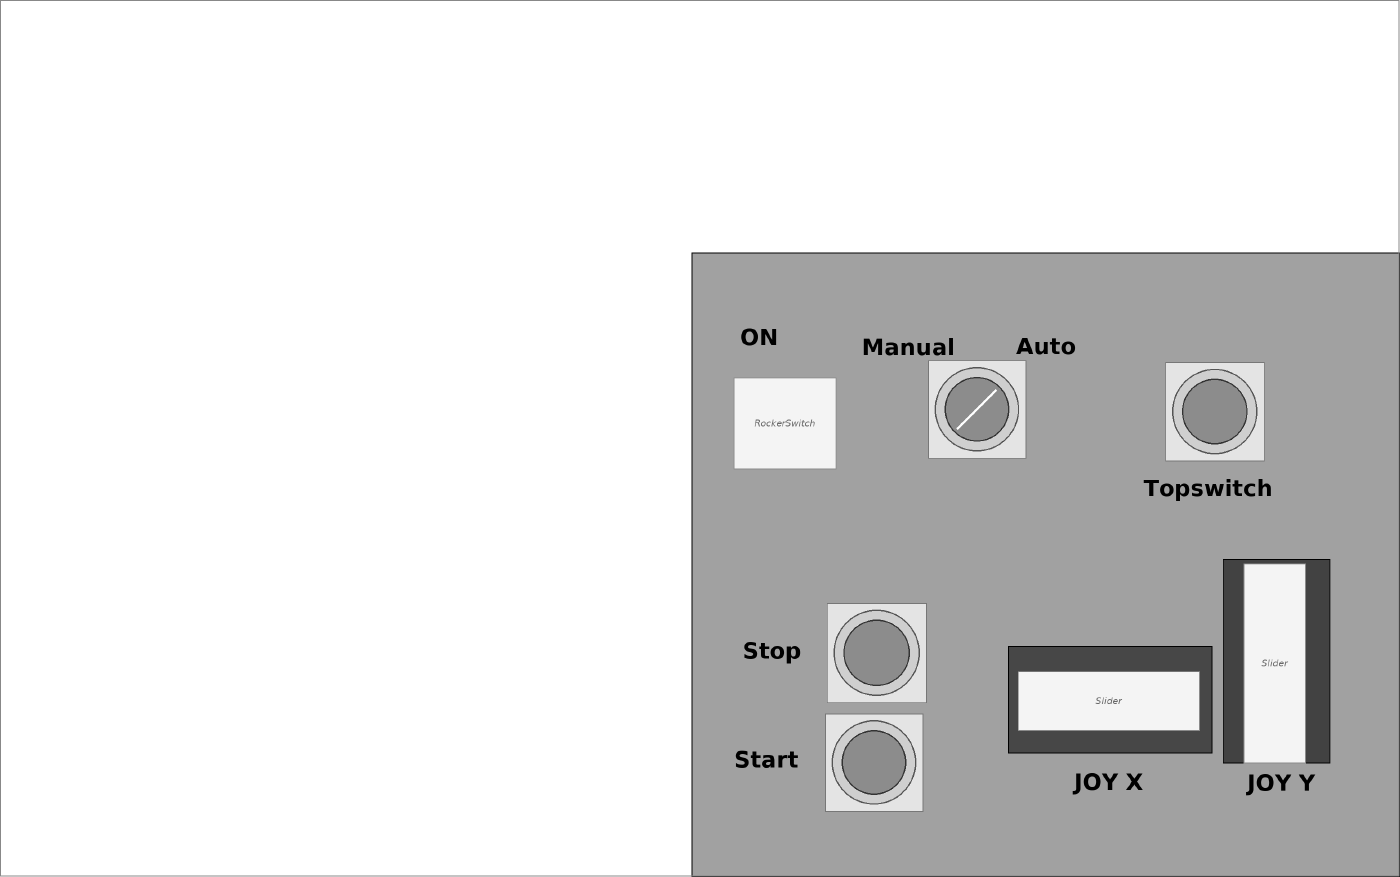
VISUALIZATION Visualization  // 1557x976
    Rectangle (769,281 788x695)
    PushSwitch (905,671 140x111), variable: task1.bStop, behaviour: TOGGLE, style: Switch-PushSwitch-Gray
    PushSwitch (908,794 128x109), variable: task1.bStart, behaviour: TOGGLE, style: Switch-PushSwitch-Gray
    Label (781,803 143x84), "Start"
    Label (787,682 143x84), "Stop"
    RockerSwitch (816,420 114x102), variable: task1.bOn, behaviour: TOGGLE, style: Switch-RockerSwitch-Gray
    RotarySwitch (1020,401 133x109), variable: task1.bManual, behaviour: TOGGLE, style: Switch-RotarySwitch-Gray
    PushSwitch (1295,403 112x110), variable: task1.bTopSwitch, behaviour: TOGGLE, style: Switch-PushSwitch-Gray
    Label (1350,856 150x30), "JOY Y"
    Label (1269,528 150x30), "Topswitch"
    Label (1158,855 150x30), "JOY X"
    RoundedRectangle (1360,622 119x227)
    Slider (1383,627 69x222), scale 0..100
    RoundedRectangle (1175,666 119x227), angle 270
    Slider (1132,747 202x66), scale 0..100
    Label (773,333 143x84), "ON"
    Label (939,344 143x84), "Manual"
    Label (1092,343 143x84), "Auto"
END_VISUALIZATION

(* stored: Version 1.1.0.1, ProductVersion 3.1.4024.12
   Visu Visualization: Id {7e46cb04-4e11-4884-a7f6-918fe33c6aed} *)
